(*
SPDX-FileCopyrightText: Â© 2026 Oleksandr Tiutyk <trofimich@gmail.com>
SPDX-License-Identifier: MIT
License: https://opensource.org/license/mit
*)

(*!
<summary>Analog output automation component converting engineering values into raw DAC signals.</summary>
<description>
Scales engineering unit values using an assigned IAnalogValueConverter and writes raw data to hardware outputs.
Successful initialization requires a parent automation component.
</description>
*)

FUNCTION_BLOCK AnalogOutput EXTENDS TOF_Automation.OutputLeafAutomationComponent
	IMPLEMENTS IAnalogOutput, TOF_Core.IIOBindable
VAR_STAT
	{attribute 'hide'} 
	_ClassName : STRING := __POUNAME();
END_VAR
VAR	
	{attribute 'hide'} 
	_RawValueType : RAW_ANALOG_VALUE_TYPE;

	{attribute 'hide'} 
	_Converter : IAnalogValueConverter;

	_CurrentValue : LREAL;
	_PreviousValue : LREAL;
	
	_RawInt16Value : REFERENCE TO INT;
	_RawInt32Value : REFERENCE TO DINT;
	_RawReal32Value : REFERENCE TO REAL; 
END_VAR

(*!
<summary>Binds component to a 16-bit signed integer output process image variable '%Q*'.</summary>
<param name="rawVariable">Reference to physical INT output variable.</param>
*)
METHOD BindToInt16IO
VAR_INPUT
	rawVariable : REFERENCE TO INT;
END_VAR
_RawValueType := RAW_ANALOG_VALUE_TYPE.INT16;

_RawInt16Value REF= rawVariable;
_RawInt32Value REF= 0;
_RawReal32Value REF= 0;
END_METHOD

(*!
<summary>Binds component to a 32-bit signed integer output process image variable '%Q*'.</summary>
<param name="rawVariable">Reference to physical DINT output variable.</param>
*)
METHOD BindToInt32IO
VAR_INPUT
	rawVariable : REFERENCE TO DINT;
END_VAR
_RawValueType := RAW_ANALOG_VALUE_TYPE.INT32;

_RawInt16Value REF= 0;
_RawInt32Value REF= rawVariable;
_RawReal32Value REF= 0;
END_METHOD

(*!
<summary>Binds component to a 32-bit float output process image variable '%Q*'.</summary>
<param name="rawVariable">Reference to physical REAL output variable.</param>
*)
METHOD BindToReal32IO
VAR_INPUT
	rawVariable : REFERENCE TO REAL;
END_VAR
_RawValueType := RAW_ANALOG_VALUE_TYPE.REAL32;

_RawInt16Value REF= 0;
_RawInt32Value REF= 0;
_RawReal32Value REF= rawVariable;
END_METHOD

(*!
<summary>Gets whether the component raw value is bound to a valid physical IO variable.</summary>
*)
{attribute 'monitoring' := 'call'}
PROPERTY FINAL BoundToIO : BOOL
GET
CASE _RawValueType OF
	RAW_ANALOG_VALUE_TYPE.INT16:
		BoundToIO := __ISVALIDREF(_RawInt16Value);
	
	RAW_ANALOG_VALUE_TYPE.INT32:
		BoundToIO := __ISVALIDREF(_RawInt32Value);
	
	RAW_ANALOG_VALUE_TYPE.REAL32:
		BoundToIO := __ISVALIDREF(_RawReal32Value);
END_CASE
END_GET
END_PROPERTY

(*!
<summary>Gets the class name of the component.</summary>
*)
{attribute 'monitoring' := 'call'}
PROPERTY ClassName : REFERENCE TO STRING
GET
ClassName REF= _ClassName;
END_GET
END_PROPERTY

(*!
<summary>Gets the assigned analog value converter.</summary>
*)
{attribute 'monitoring' := 'call'}
PROPERTY FINAL Converter : IAnalogValueConverter
GET
Converter := _Converter;
END_GET
END_PROPERTY

(*!
<summary>Initializes component name, parent and converter dependency.</summary>
<param name="bInitRetains">TRUE: retain variables are initialized.</param>
<param name="bInCopyCode">TRUE: instance copied to copy code (online change).</param>
<param name="name">Component instance name.</param>
<param name="parent">Nonzero parent automation component required for successful Initialize().</param>
<param name="converter">Mandatory analog value converter dependency.</param>
*)
METHOD FB_init : BOOL
VAR_INPUT
	bInitRetains : BOOL; // TRUE: the retain variables are initialized (reset warm / reset cold)
	bInCopyCode : BOOL;  // TRUE: the instance will be copied to the copy code afterward (online change)
	name : WSTRING;
	parent : TOF_Automation.IParentAutomationComponent;
	converter : IAnalogValueConverter;
END_VAR
IF NOT bInCopyCode THEN
	_Converter := converter;
END_IF
END_METHOD

(*!
<summary>Gets the namespace name of the component.</summary>
*)
{attribute 'monitoring' := 'call'}
PROPERTY NamespaceName : REFERENCE TO STRING
GET
NamespaceName REF= CurrentNamespace.Name;
END_GET
END_PROPERTY

(*!
<summary>Validates that mandatory converter dependency is configured.</summary>
*)
METHOD PROTECTED OnInitializing : BOOL
IF _Converter = 0 THEN
	TOF_Core.Exceptions.ThrowClassInitialization(
		sourceNamespaceName := NamespaceName,
		sourceClassName := ClassName,
		sourcePOUName := __POUNAME(),
		sourcePosition := __POSITION(),
		errorMessage := "converter not specified"
	);
END_IF

OnInitializing := TRUE;
END_METHOD

(*!
<summary>Scales engineering value to raw DAC signal and writes to bound hardware output.</summary>
*)
METHOD PROTECTED OnProcessOutput
setRawValueByUnion(
	_Converter.ConvertAnalogValueToRawValue(
		analogValue := _CurrentValue,
		rawValueType := _RawValueType
	)
);

_PreviousValue := _CurrentValue;
END_METHOD

(*!
<summary>Gets current raw hardware DAC value cast to LREAL.</summary>
*)
{attribute 'monitoring' := 'call'}
PROPERTY FINAL RawValue : LREAL
GET
CASE _RawValueType OF
	RAW_ANALOG_VALUE_TYPE.INT16:
		RawValue := SEL(__ISVALIDREF(_RawInt16Value), 0, TO_LREAL(_RawInt16Value));
	
	RAW_ANALOG_VALUE_TYPE.INT32:
		RawValue := SEL(__ISVALIDREF(_RawInt32Value), 0, TO_LREAL(_RawInt32Value));
	
	RAW_ANALOG_VALUE_TYPE.REAL32:
		RawValue := SEL(__ISVALIDREF(_RawReal32Value), 0, TO_LREAL(_RawReal32Value));
END_CASE
END_GET
END_PROPERTY

(*!
<summary>Gets the raw analog data representation type.</summary>
*)
{attribute 'monitoring' := 'call'}
PROPERTY FINAL RawValueType : RAW_ANALOG_VALUE_TYPE
GET
RawValueType := _RawValueType;
END_GET
END_PROPERTY

(*!
<summary>Gets the memory size of the instance.</summary>
*)
{attribute 'monitoring' := 'call'}
PROPERTY SelfSize : ULINT
GET
SelfSize := XSIZEOF(THIS^);
END_GET
END_PROPERTY

METHOD PRIVATE setRawValueByUnion
VAR_INPUT
	rawValueUnion : RAW_ANALOG_VALUE;
END_VAR
CASE _RawValueType OF
	RAW_ANALOG_VALUE_TYPE.INT16:
		IF __ISVALIDREF(_RawInt16Value) THEN
			_RawInt16Value := rawValueUnion.Int16; 
		END_IF
	
	RAW_ANALOG_VALUE_TYPE.INT32:
		IF __ISVALIDREF(_RawInt32Value) THEN
			_RawInt32Value := rawValueUnion.Int32; 
		END_IF
	
	RAW_ANALOG_VALUE_TYPE.REAL32:
		IF __ISVALIDREF(_RawReal32Value) THEN
			_RawReal32Value := rawValueUnion.Real32; 
		END_IF
END_CASE
END_METHOD

(*!
<summary>Gets or sets engineering unit value to output.</summary>
*)
{attribute 'monitoring' := 'call'}
PROPERTY Value : LREAL
GET
Value := _CurrentValue;
END_GET
SET
_CurrentValue := Value;
END_SET
END_PROPERTY

END_FUNCTION_BLOCK

(* stored: Version 1.1.0.1
   POU AnalogOutput: Id {2baa0bb5-149e-4c48-8457-b1d26d365163}, SpecialFunc None
   Folder Overriden members: Id {ad93e144-ffa3-4723-86ea-fe15cc56a4b8}
   Folder Service members: Id {d31b0d7d-549a-4487-ad09-1fd6e7696561}
   Method BindToInt16IO: Id {ea1538b8-fa62-4d20-afa4-4702479ecd66}
   Method BindToInt32IO: Id {d1d29b44-661e-4f10-b84c-c81909342e2c}
   Method BindToReal32IO: Id {215b589f-5793-430e-aff2-f6be3317608a}
   Property BoundToIO: Id {b4ad226a-23ac-46e8-91eb-1763c4519e6b}
   Get Get: Id {56dea10f-be64-4327-8f8a-c42fa9fed1fc}
   Property ClassName: Id {27685b38-d546-4e7a-a9dd-88ead7d46659}
   Get Get: Id {8e787df8-fc1d-499a-a442-3dee7862ab93}
   Property Converter: Id {ee5e3166-f8c8-47de-8453-11334cbecf1b}
   Get Get: Id {1dd401e0-3fb3-4aec-9bb3-411f7744b3f5}
   Method FB_init: Id {a9f49d33-e9ea-4be3-bd71-06a12d50e73a}
   Property NamespaceName: Id {1b722dcb-bc0b-4369-815d-7d25318c6696}
   Get Get: Id {ed0ba56c-ca57-4831-a069-b096cb8b456d}
   Method OnInitializing: Id {e669a5ff-36c0-4fd0-81b0-71f5545efcf0}
   Method OnProcessOutput: Id {7a765b44-1dba-42c2-8447-7ae0226f3069}
   Property RawValue: Id {d565d9b5-3dcf-4ebc-8d53-c6e13619f73d}
   Get Get: Id {9b5db42e-eece-4bbf-8b70-0e27ec9bf3ce}
   Property RawValueType: Id {0069a9c5-d054-488f-b70f-c7c629a45667}
   Get Get: Id {d7eaf920-e53f-4eda-a319-b1b80f0627b1}
   Property SelfSize: Id {13ce6ab1-facb-4c54-bd07-b636d694c444}
   Get Get: Id {afe2b91b-981a-42f5-b330-ccfe8915f117}
   Method setRawValueByUnion: Id {b2e6cda0-d593-45d0-b846-0c65d7e2e34f}
   Property Value: Id {f20d1a0d-5f58-46d7-b903-483c9d1e4968}
   Get Get: Id {1f0cbb7d-0f9c-449f-bc90-8e9af89a0352}
   Set Set: Id {afec2ca8-e3f7-4ca0-b4c8-23b143028807} *)
